(* IEC 61131-3 sources: industrial-simulator/plc/openplc, 2 files *)

(* ---- conveyor.st ---- *)
(* Industrial Simulator - programme de demonstration Phase 3
   Machine : convoyeur_01 (usine : simulator/config/factory.json)

   Logique d'automatisme exigee par le cahier des charges :
     SI sensor_entry = TRUE  ALORS conveyor.run = TRUE
     SI sensor_exit  = TRUE  ALORS conveyor.run = FALSE

   Adressage (slave device "simulateur" declare dans OpenPLC) :
     %IX100.0 <- discrete input 0 du simulateur (sensor_entry)
     %IX100.1 <- discrete input 1 du simulateur (sensor_exit)
     %QX100.0 -> coil 0 du simulateur (conveyor_01.run)

   NB important : OpenPLC range les E/S des devices distants a partir de
   %I/%Q100 (voir updateBuffersIn_MB dans core/modbus_master.cpp) ; la bande
   basse (%I0/%Q0) est reservee a l'image de son propre serveur Modbus.

   Le maintien de la marche (memoire SET/RESET) est assure par ces deux
   affectations : conveyor_run garde sa valeur tant qu'aucun capteur n'agit.
   C'est la logique d'automatisme, elle vit dans le PLC, pas dans le simulateur.

   OpenPLC v3 exige un programme IEC 61131-3 complet : PROGRAM + CONFIGURATION.
   La tache Main est executee toutes les 50 ms ; la scrutation Modbus du
   simulateur est reglee cote OpenPLC (Slave_polling, defaut 100 ms). *)

PROGRAM prog0
  VAR
    sensor_entry AT %IX100.0 : BOOL;
    sensor_exit AT %IX100.1 : BOOL;
    conveyor_run AT %QX100.0 : BOOL;
  END_VAR

  IF sensor_entry THEN
    conveyor_run := TRUE;    (* capteur d'entree : marche *)
  END_IF;

  IF sensor_exit THEN
    conveyor_run := FALSE;   (* capteur de sortie : arret *)
  END_IF;
END_PROGRAM

CONFIGURATION Config0

  RESOURCE Res0 ON PLC
    TASK Main(INTERVAL := T#50ms,PRIORITY := 0);
    PROGRAM Inst0 WITH Main : prog0;
  END_RESOURCE
END_CONFIGURATION

(* ---- conveyor_cycle.st ---- *)
(* Industrial Simulator - Phase 4 : cycle continu
   Variante du programme convoyeur : la boite ne reste pas bloquee au
   capteur de sortie ; apres 2 s de pause, le convoyeur l'evacue, puis
   se remet en attente de la boite suivante.

   Sequence (GRAFCET equivalent) :
     ATTENTE --entree--> MARCHE --capteur sortie--> ARRET(2s)
     ARRET --2s--> EVACUATION --boite liberee + 1s--> ATTENTE

   Adressage identique a conveyor.st (bande %I/%Q100 des devices distants). *)

PROGRAM prog0
  VAR
    sensor_entry AT %IX100.0 : BOOL;
    sensor_exit AT %IX100.1 : BOOL;
    conveyor_run AT %QX100.0 : BOOL;
  END_VAR
  VAR
    (* NB : ce matiec refuse de melanger variables AT et variables internes
       dans un meme bloc VAR - d'ou les deux blocs. *)
    pause_ton : TON;      (* delai d'arret sur le capteur de sortie *)
    tail_ton : TON;       (* delai d'evacuation apres liberation du capteur *)
    evacuating : BOOL;
  END_VAR

  (* Marche / arret nominaux *)
  IF sensor_entry AND NOT evacuating THEN
    conveyor_run := TRUE;
  END_IF;

  IF sensor_exit THEN
    conveyor_run := FALSE;
  END_IF;

  (* Apres 2 s posee sur le capteur de sortie : evacuer *)
  pause_ton(IN := sensor_exit, PT := T#2s);
  IF pause_ton.Q THEN
    evacuating := TRUE;
  END_IF;

  IF evacuating THEN
    conveyor_run := TRUE;
    (* la boite a quitte le capteur : encore 1 s pour la faire tomber au bout *)
    tail_ton(IN := NOT sensor_exit, PT := T#1s);
    IF tail_ton.Q THEN
      conveyor_run := FALSE;
      evacuating := FALSE;
    END_IF;
  END_IF;
END_PROGRAM

CONFIGURATION Config0

  RESOURCE Res0 ON PLC
    TASK Main(INTERVAL := T#50ms,PRIORITY := 0);
    PROGRAM Inst0 WITH Main : prog0;
  END_RESOURCE
END_CONFIGURATION
